{attribute 'pack_mode' := '1'}
TYPE ST_Command :
STRUCT
 ProtocolVersion, ProfileFingerprint : UDINT;
 Enable, Disable, Reset, Stop : BYTE;
 Mode : INT;
 TorqueNm, RampNmPerSec, PowerW : LREAL;
 Heartbeat : UDINT;
END_STRUCT
END_TYPE

(* stored: Version 1.1.0.1, ProductVersion 3.1.4024.0
   DUT ST_Command: Id {00000000-0000-4000-8000-000000000001} *)
